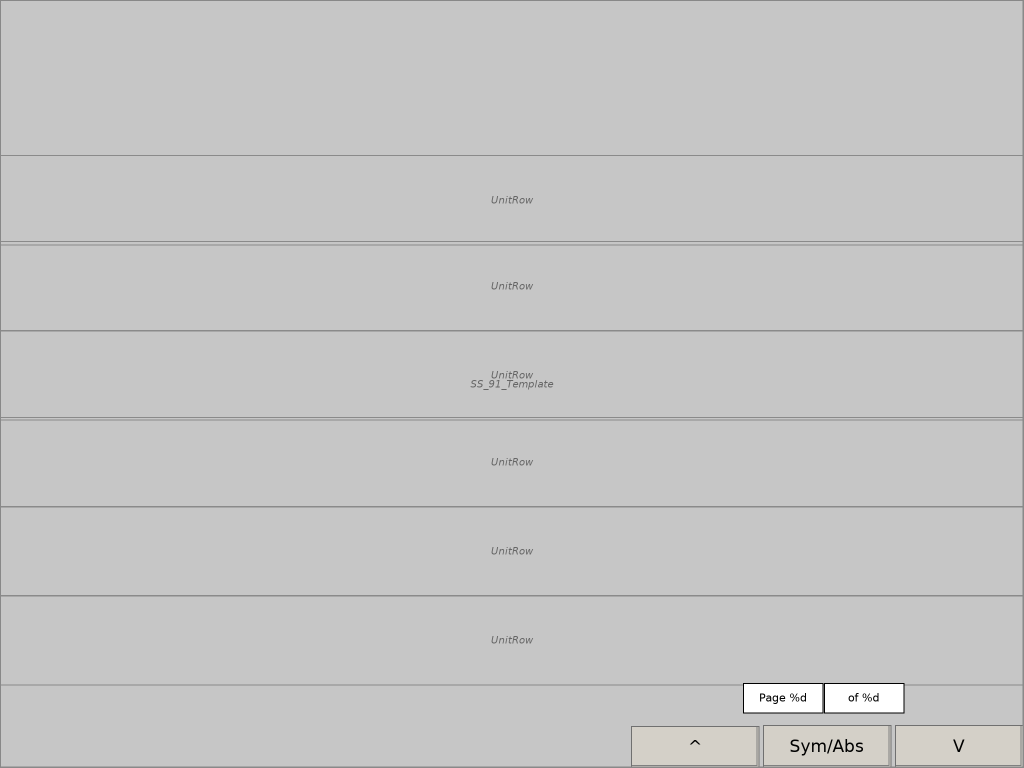
VISUALIZATION Mc_01_Units  // 1024x768
    Frame (0,0 1024x768)
        shows SS_91_Template()
    Frame (0,155 1024x90)
        shows UnitRow(MotionRowInstanceSingle := HMIData.gUnitRows.gMotionRow1, MotionRowButtonsSingle := HMIData.gUnitButtons.gMotionRow1btn)
    Frame (0,241 1024x90)
        shows UnitRow(MotionRowInstanceSingle := HMIData.gUnitRows.gMotionRow2, MotionRowButtonsSingle := HMIData.gUnitButtons.gMotionRow2btn)
    Frame (0,330 1024x90)
        shows UnitRow(MotionRowInstanceSingle := HMIData.gUnitRows.gMotionRow3, MotionRowButtonsSingle := HMIData.gUnitButtons.gMotionRow3btn)
    Frame (0,417 1024x90)
        shows UnitRow(MotionRowInstanceSingle := HMIData.gUnitRows.gMotionRow4, MotionRowButtonsSingle := HMIData.gUnitButtons.gMotionRow4btn)
    Frame (0,506 1024x90)
        shows UnitRow(MotionRowInstanceSingle := HMIData.gUnitRows.gMotionRow5, MotionRowButtonsSingle := HMIData.gUnitButtons.gMotionRow5btn)
    Frame (0,595 1024x90)
        shows UnitRow(MotionRowInstanceSingle := HMIData.gUnitRows.gMotionRow6, MotionRowButtonsSingle := HMIData.gUnitButtons.gMotionRow6btn)
    Button (763,725 128x42), "Sym/Abs", colour toggle: HMIData.btnAbsMode
        toggle HMIData.btnAbsMode
    Button (631,726 128x41), "^"
        tap HMIData.btnPrevPage
    Button (895,725 128x42), "V"
        tap HMIData.btnNextPage
    Rectangle (743,683 80x30), "Page %d", text variable: HMIData.gActivePageNumber
    Rectangle (824,683 80x30), "of %d", text variable: HMIData.gMaxPageNumber
END_VISUALIZATION

(* stored: Version 1.1.0.1, ProductVersion 3.1.4024.12
   Visu Mc_01_Units: Id {568f4bda-c6d5-45bc-bae5-d7f9fed8a64f} *)
